Staubli VAL3: type.pgx

public program type(num pX (dimensions=1), num pY (dimensions=1), string pStr (dimensions=1))
begin
  //---------------------------------
  //  S H O W   O N E   S T R I N G
  //---------------------------------
  // Display one string to pX column
  // and pY Line
  //
  gotoxy(pX,pY)
  put(pStr)
end
